(* Logix 5000 project; controller EuniceF_Lab2 vendor 1 type 14 code 150 rev 37.11; software revision 37.00 *)

TASK MainTask (continuous, watchdog 500 ms) : MainProgram

MODULES
   Local : vendor 1 type 14 code 150 (Compact 0, rev 37.11)
      Discrete_IO : Embedded (Compact 1, rev 3.1, Output RPI 20 ms)
      Analog_IO : Embedded (Compact 2, rev 1.1, Output RPI 80 ms)
      Counters : Embedded (Compact 3, rev 1.1, Output RPI 20 ms)
END_MODULES

VAR_GLOBAL   (* controller tags *)
   Diif_Pressure : ALIAS FOR Local:2:I.Ch3Data;
   DrainValve : ALIAS FOR Local:1:O.Data.10;
   Mixer : ALIAS FOR Local:1:O.Data.9;
   Pump : ALIAS FOR Local:1:O.Data.8;
   Start : ALIAS FOR Local:1:I.Data.11;
   Stop : ALIAS FOR Local:1:I.Data.9;
   T1 : TIMER := (PRE := 10000);
   Valve_Position : ALIAS FOR Local:2:O.Ch1Data;
END_VAR

PROGRAM MainProgram   (* main routine MainRoutine *)

ROUTINE MainRoutine   (* ladder *)
   0: ;
END_ROUTINE
END_PROGRAM
